Fanuc KAREL source: ko00039.KL

-- PROVISIONAL review KL for V1013-1; original PC SHA256 2b8ca6d92ee89e51487eb9f949f7217f4df56945c97bfba67883ca110bb98a91
-- Incomplete behavior may be omitted. Consult companion uncertainty JSON. Do not deploy.
PROGRAM KO00039
%NOLOCKGROUP
BEGIN
  -- UNRESOLVED_PC offsets 5-12; opcodes 9D,23
  -- UNRESOLVED_PC offsets 17-69; opcodes 27,27,49,7E,AD,27,49,7E,AD,22,31,7E,4A
  -- UNRESOLVED_PC offsets 74-78; opcodes 7F
END KO00039
